# EPICS autosave request: iocBoot/iocAmptek/auto_settings.req
file "mca_settings.req",          P=$(P), M=mca1
